(* This function is for the Cold Cathode MKS 500 connected to Beckhoff EP boxes.
A separate function block is necessary for the MKS500-to-EP box interface beacuse the EP
boxes do not natively support the 5v IO signals on the MKS500 gauge.*)
(*This function provides ILK and Set Point Protection for the Cold Cathode*)
(* 500 Logarithmic Output Conversion, factory default configuration *)
FUNCTION_BLOCK FB_MKS500_EP
VAR_IN_OUT
		
END_VAR
VAR_INPUT

	PG	:	ST_VG;
END_VAR
VAR_OUTPUT
{attribute 'pytmc' := '
    pv: 
	'}
	IG : ST_VG;
END_VAR
VAR
	rV : REAL;
	pBase : REAL :=1.0E-10;//default curve base pressure is 1E-10. Confusing since can't actually read that low using analog out.
	vBase : REAL := 0; // corresponding vbase 0V based on default curve.  See manual pg. 44
	vSlope : REAL := 1.0; //looks correct for default curve
	GaugeTurnOnTmr : TON;
	MinPressure: REAL := 1E-10;
	cDefaultPressure : REAL := 0;
	
	
	(*IOs to be linked*)
	/// Controls and I/Os
	i_iPRESS_R AT %I* :INT; // input Pressure // Link to analog Input
	q_xHV_DIS AT %Q* : BOOL; // Enable High Voltage when True // 'TcLinkTo' (EP2624) ^Output
	//
END_VAR

(* 500 Logarithmic Output Conversion, factory default configuration *)


(*check health of the ethercat terminal*)

rV := 10*INT_TO_REAL(IG.i_iPRESS_R)/32767;

(* Set Guage State based on the inputs HV ON and Discharge current*)
IF rV >= 0.49 AND rV < 0.6  THEN
	IG.eState := Starting;
	IG.rPRESS := LREAL_TO_REAL(EXPT(10,((rV-vBase)/vSlope+LOG(pBase))));
ELSE
	IG.eState := Valid;
	IG.rPRESS := LREAL_TO_REAL(EXPT(10,((rV-vBase)/vSlope+LOG(pBase))));
END_IF



(* Ion Gauge Protection Functions *)
(* If the PG pressure is greater than the VG.PRO_SP then the gauge is disabled *)
(* If the PG pressure is less than the VG.PRO_SP then the gauge is enabled *)
(* This FB also implements some hysteresis so the gauge doesn't have rapid power cycling while near the turn on boundary *)



IF PG.rPRESS <= IG.rPRO_SP AND PG.xPRESS_OK THEN

	IG.q_xHV_DIS := IG.xHV_SW;
	IG.xILKOk := TRUE;
ELSIF IG.q_xHV_DIS THEN
	IF IG.rPRESS > (IG.rPRO_SP + IG.rHYS_PR)  OR PG.rPRESS > (IG.rPRO_SP + IG.rHYS_PR) THEN
		IG.q_xHV_DIS := FALSE;
		IG.xHV_SW := FALSE;
	END_IF
ELSE
	IG.q_xHV_DIS := FALSE;
	IG.xHV_SW := FALSE;
	IG.xILKOk := FALSE;
END_IF

(* Pressure gauge OK checks *)

GaugeTurnOnTmr(IN:=IG.q_xHV_DIS, PT:=T#10S, Q=>IG.xTurnOnTime);


//Backwards compatibility
IG.xPRESS_OK := (IG.eState = Valid) OR IG.xBAKEOUT;

(* Setpoint evaluation *)
IG.xAT_VAC := (IG.xPRESS_OK AND (IG.rPRESS < IG.rVAC_SP)) OR IG.xBAKEOUT AND (IG.eState = Valid) ;


(*Soft IO Linking*)
// check ethercat Diagnostics
IO();

ACTION IO:
(*soft link inputs*)
IG.i_iPRESS_R:=	i_iPRESS_R; 
(*soft link outputs*)
q_xHV_DIS := IG.q_xHV_DIS;
END_ACTION

METHOD M_HVE : BOOL
VAR_INPUT
		enable:bool; // set to true to enable, false to disable;
END_VAR

this^.IG.xHV_SW:= NOT(enable);
END_METHOD

END_FUNCTION_BLOCK

(* stored: Version 1.1.0.1, ProductVersion 3.1.4024.2
   POU FB_MKS500_EP: Id {4da1e942-f359-4f6e-ab12-d5a0031e68e6}, SpecialFunc None
   Action IO: Id {8ad71ac6-f961-40c8-a3be-ad3367f81f67}
   Method M_HVE: Id {5c5dd30f-1cf9-426d-9ab9-5103df771146} *)
